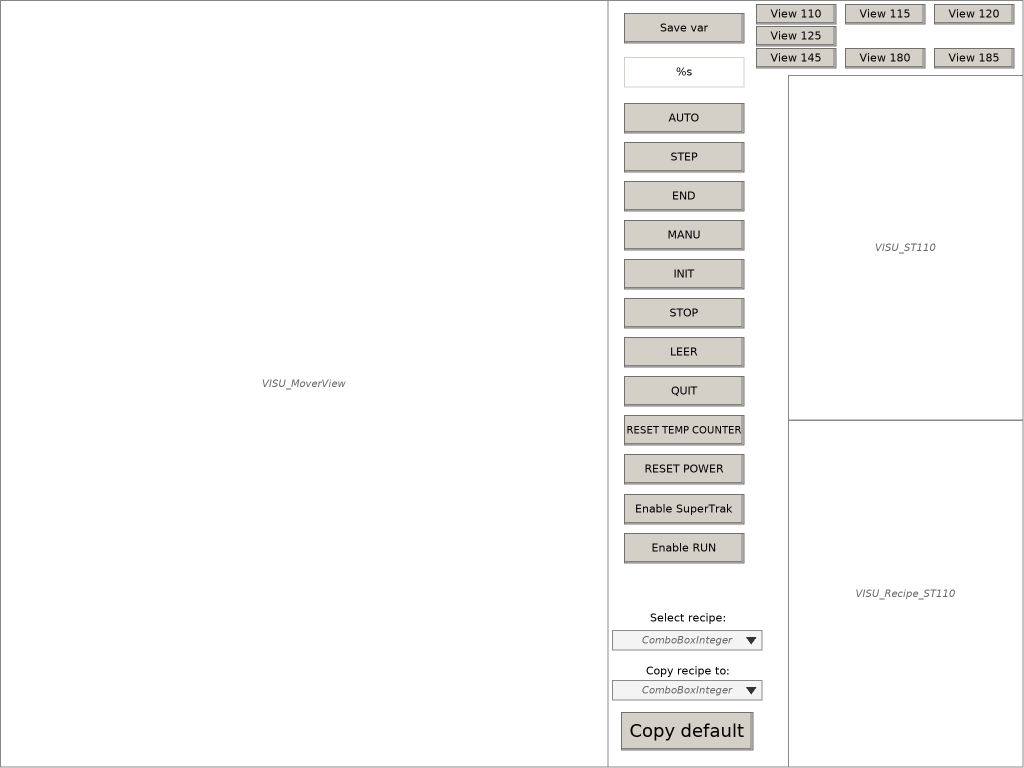
VISUALIZATION VISU_main  // 1024x768
    TabControl (0,0 608x767)
        shows VISU_MoverView()
        shows VISU_LinearConfigArray()
        shows VISU_MoverDetail()
        shows VISU_Cylinder2PosConfig()
        [0]: TabTitle=Mover Track, ImageId=Custom.Shuttle Full
        [1]: TabTitle=Linear Axis, ImageId=Custom.RotTable_3Slots
        [2]: TabTitle=Mover details
        [3]: TabTitle=Cylinder config
    Button (624,103 120x30), "AUTO", colour toggle: HMI.btArMain[0].on, input disabled if: HMI.btArMain[0].disable
        tap HMI.btArMain[0].button
    Button (624,142 120x30), "STEP", colour toggle: HMI.btArMain[1].on, input disabled if: HMI.btArMain[1].disable
        tap HMI.btArMain[1].button
    Button (624,181 120x30), "END", colour toggle: HMI.btArMain[2].on, input disabled if: HMI.btArMain[2].disable
        tap HMI.btArMain[2].button
    Button (624,259 120x30), "INIT", colour toggle: HMI.btArMain[4].on, input disabled if: HMI.btArMain[4].disable
        tap HMI.btArMain[4].button
    Button (624,298 120x30), "STOP", colour toggle: HMI.btArMain[5].disable, input disabled if: HMI.btArMain[5].disable
        tap HMI.btArMain[5].button
    Button (624,337 120x30), "LEER", colour toggle: HMI.btArMain[6].disable, input disabled if: HMI.btArMain[6].disable
        tap HMI.btArMain[6].button
    Button (624,376 120x30), "QUIT", colour toggle: HMI.btArMain[7].disable, input disabled if: HMI.btArMain[7].disable
        tap HMI.btArMain[7].button
    Button (624,415 120x30), "RESET TEMP COUNTER", colour toggle: HMI.btArMain[8].disable, input disabled if: HMI.btArMain[8].disable
        tap HMI.btArMain[8].button
    Button (624,220 120x30), "MANU", colour toggle: HMI.btArMain[3].on, input disabled if: HMI.btArMain[3].disable
        tap HMI.btArMain[3].button
    Textfield (624,57 120x30), "%s", text variable: _14_STATE.sStateDbg
    Button (624,454 120x30), "RESET POWER"
        tap HMI.Tast_BL
    Button (624,13 120x30), "Save var", input disabled if: TRUE
        tap FileMan.bSaveData
    Frame (788,75 235x345)
        shows VISU_ST110()
        shows VISU_ST115()
        shows VISU_ST120()
        shows VISU_ST125()
        shows VISU_ST145()
        shows VISU_ST180()
        shows VISU_ST185()
    Button (845,4 80x20), "View 115"
        OnMouseDown: FrameSelectionChange Selection=SelectedFrame=06e07b94-3d2f-4429-a7a0-840881734514, Selection=1, GlobSel=AssignType=Directly, SelType=Locally
        OnMouseDown: FrameSelectionChange Selection=SelectedFrame=9156b980-1735-4d37-9321-1bea537ecf5c, Selection=1, GlobSel=AssignType=Directly, SelType=Locally
    Button (756,4 80x20), "View 110"
        OnMouseDown: FrameSelectionChange Selection=SelectedFrame=06e07b94-3d2f-4429-a7a0-840881734514, GlobSel=AssignType=Directly, SelType=Locally
        OnMouseDown: FrameSelectionChange Selection=SelectedFrame=9156b980-1735-4d37-9321-1bea537ecf5c, GlobSel=AssignType=Directly, SelType=Locally
    Button (934,4 80x20), "View 120"
        OnMouseDown: FrameSelectionChange Selection=SelectedFrame=06e07b94-3d2f-4429-a7a0-840881734514, Selection=2, GlobSel=AssignType=Directly, SelType=Locally
        OnMouseDown: FrameSelectionChange Selection=SelectedFrame=9156b980-1735-4d37-9321-1bea537ecf5c, Selection=2, GlobSel=AssignType=Directly, SelType=Locally
    Frame (788,420 235x347)
        shows VISU_Recipe_ST110()
        shows VISU_Recipe_ST115()
        shows VISU_Recipe_ST120()
        shows VISU_Recipe_ST125()
        shows VISU_Recipe_ST145()
        shows VISU_Recipe_ST180()
        shows VISU_Recipe_ST185()
    Button (756,26 80x20), "View 125"
        OnMouseDown: FrameSelectionChange Selection=SelectedFrame=06e07b94-3d2f-4429-a7a0-840881734514, Selection=3, GlobSel=AssignType=Directly, SelType=Locally
        OnMouseDown: FrameSelectionChange Selection=SelectedFrame=9156b980-1735-4d37-9321-1bea537ecf5c, Selection=3, GlobSel=AssignType=Directly, SelType=Locally
    Button (624,494 120x30), "Enable SuperTrak", colour toggle: gMoverAxis.Q_CT_Track_to_BR.asStruct.bCommand.0
        toggle gMoverAxis.Q_CT_Track_to_BR.asStruct.bCommand.0
    Button (624,533 120x30), "Enable RUN", colour toggle: gMoverAxis.Q_CT_Track_to_BR.asStruct.bCommand.2
        toggle gMoverAxis.Q_CT_Track_to_BR.asStruct.bCommand.2
    ComboBoxInteger (612,630 150x20), variable: PERS.eRecipeCurrent
    Label (613,661 150x20), "Copy recipe to:"
    ComboBoxInteger (612,680 150x20), variable: _20_AUTO.iRecipeCopyDest
    Button (621,712 132x38), "Copy default"
        tap HMI.btCopyRecipe.button
    Button (756,48 80x20), "View 145"
        OnMouseDown: FrameSelectionChange Selection=SelectedFrame=06e07b94-3d2f-4429-a7a0-840881734514, Selection=4, GlobSel=AssignType=Directly, SelType=Locally
        OnMouseDown: FrameSelectionChange Selection=SelectedFrame=9156b980-1735-4d37-9321-1bea537ecf5c, Selection=4, GlobSel=AssignType=Directly, SelType=Locally
    Label (613,608 150x20), "Select recipe:"
    Button (845,48 80x20), "View 180"
        OnMouseDown: FrameSelectionChange Selection=SelectedFrame=06e07b94-3d2f-4429-a7a0-840881734514, Selection=5, GlobSel=AssignType=Directly, SelType=Locally
        OnMouseDown: FrameSelectionChange Selection=SelectedFrame=9156b980-1735-4d37-9321-1bea537ecf5c, Selection=5, GlobSel=AssignType=Directly, SelType=Locally
    Button (934,48 80x20), "View 185"
        OnMouseDown: FrameSelectionChange Selection=SelectedFrame=06e07b94-3d2f-4429-a7a0-840881734514, Selection=6, GlobSel=AssignType=Directly, SelType=Locally
        OnMouseDown: FrameSelectionChange Selection=SelectedFrame=9156b980-1735-4d37-9321-1bea537ecf5c, Selection=6, GlobSel=AssignType=Directly, SelType=Locally
END_VISUALIZATION

(* stored: Version 1.1.0.1, ProductVersion 3.1.4024.6
   Visu VISU_main: Id {d72905fe-72a6-4ef2-acdb-6547139e7766} *)
